{attribute 'qualified_only'}
{attribute 'strict'}
TYPE EExpressionType :
(
	none := 0,
	boolean := 1,
	comparison := 2,
	value := 3
);
END_TYPE

(* stored: Version 1.1.0.1, ProductVersion 3.1.4024.9
   DUT EExpressionType: Id {87d49123-8fc9-4335-81f4-6b753bdfbff8} *)
